Staubli VAL3: CartesianPos.dtx

public pointRx CartesianPos = {fatherId=world[0]}
